FUNCTION_BLOCK PICKER_MODEL_NO_SFC_VIEW (* Composite Function Block Type *)
  (* Standard: 61499-2 *)
  (* Version 0.2, 2003-12-05, JHC, Rockwell Automation, Renamed from NEWCOMPFB. *)
  (* Version 0.1, 2002-01-08, JHC, Rockwell Automation, Added DLY FB as example. *)
  (* Version 0.0, 2000-05-27, JHC, Rockwell Automation *)
  (* Compiler header: package fb.rt.pnp; *)
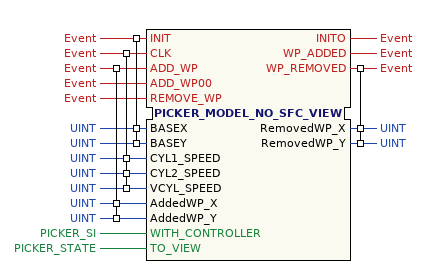
  EVENT_INPUT
    INIT WITH BASEX, BASEY; (* Initialisation *)
    CLK WITH CYL1_SPEED, CYL2_SPEED, VCYL_SPEED;
    ADD_WP WITH AddedWP_X, AddedWP_Y;
    ADD_WP00;
    REMOVE_WP;
  END_EVENT
  EVENT_OUTPUT
    INITO; (* Initialization Confirm *)
    WP_ADDED;
    WP_REMOVED WITH RemovedWP_X, RemovedWP_Y;
  END_EVENT
  VAR_INPUT
    BASEX : UINT;
    BASEY : UINT;
    CYL1_SPEED : UINT;
    CYL2_SPEED : UINT;
    VCYL_SPEED : UINT;
    AddedWP_X : UINT;
    AddedWP_Y : UINT;
  END_VAR
  VAR_OUTPUT
    RemovedWP_X : UINT;
    RemovedWP_Y : UINT;
  END_VAR
  SOCKETS
    WITH_CONTROLLER : PICKER_SI;
    TO_VIEW : PICKER_STATE;
  END_SOCKETS
  FBS
    MODEL : Model;
    s11 : my_sensor(ZONE := [305,310]);
    s12 : my_sensor(ZONE := [381,385]);
    s13 : my_sensor(ZONE := [455,460]);
    s14 : my_sensor(ZONE := [535,540]);
    Machado_SFC : MachadoSFC;
  END_FBS
  EVENT_CONNECTIONS
    INIT TO MODEL.INIT;
    MODEL.INITO TO TO_VIEW.INIT;
    MODEL.INITO TO INITO;
    MODEL.CNF TO WITH_CONTROLLER.CNF;
    WITH_CONTROLLER.REQ TO MODEL.REQ;
    CLK TO MODEL.CLK;
    ADD_WP TO MODEL.ADD_WP;
    REMOVE_WP TO MODEL.REMOVE_WP;
    MODEL.WP_ADDED TO WP_ADDED;
    MODEL.WP_REMOVED TO WP_REMOVED;
    MODEL.INITO TO s11.INIT;
    s11.INITO TO s12.INIT;
    s12.INITO TO s13.INIT;
    s13.INITO TO s14.INIT;
    MODEL.CNF TO s11.REQ;
    MODEL.CNF TO s12.REQ;
    MODEL.CNF TO s13.REQ;
    MODEL.CNF TO s14.REQ;
    s11.CNF TO WITH_CONTROLLER.CNF;
    s12.CNF TO WITH_CONTROLLER.CNF;
    s13.CNF TO WITH_CONTROLLER.CNF;
    s14.CNF TO WITH_CONTROLLER.CNF;
    ADD_WP00 TO MODEL.ADD_WP00;
    s14.INITO TO Machado_SFC.INIT;
    MODEL.CHG TO Machado_SFC.REQ;
    MODEL.CHG TO WITH_CONTROLLER.CNF;
    MODEL.CNF TO TO_VIEW.CHG;
    s11.CNF TO Machado_SFC.REQ;
    s12.CNF TO Machado_SFC.REQ;
    s13.CNF TO Machado_SFC.REQ;
    s14.CNF TO Machado_SFC.REQ;
    Machado_SFC.CNF TO MODEL.CYL_IND;
  END_CONNECTIONS
  DATA_CONNECTIONS
    MODEL.BASE_X TO TO_VIEW.BASE_X;
    MODEL.BASE_Y TO TO_VIEW.BASE_Y;
    MODEL.CYL1_X TO TO_VIEW.CYL1_X;
    MODEL.CYL1_Y TO TO_VIEW.CYL1_Y;
    MODEL.CYL2_X TO TO_VIEW.CYL2_X;
    MODEL.CYL2_Y TO TO_VIEW.CYL2_Y;
    MODEL.VCYL_X TO TO_VIEW.VCYL_X;
    MODEL.VCYL_Y TO TO_VIEW.VCYL_Y;
    MODEL.WP_X TO TO_VIEW.WP1_X;
    MODEL.WP_Y TO TO_VIEW.WP1_Y;
    MODEL.VACUUM_ON TO TO_VIEW.VACUUM_ON;
    BASEX TO MODEL.BASEX;
    BASEY TO MODEL.BASEY;
    CYL1_SPEED TO MODEL.CYL1_SPEED;
    CYL2_SPEED TO MODEL.CYL2_SPEED;
    VCYL_SPEED TO MODEL.VCYL_SPEED;
    MODEL.vchome TO WITH_CONTROLLER.vchome;
    MODEL.vcend TO WITH_CONTROLLER.vcend;
    AddedWP_X TO MODEL.AddedWP_X;
    AddedWP_Y TO MODEL.AddedWP_Y;
    MODEL.RemovedWP_X TO RemovedWP_X;
    MODEL.RemovedWP_Y TO RemovedWP_Y;
    MODEL.VCYL_X TO s11.POS;
    MODEL.VCYL_X TO s12.POS;
    MODEL.VCYL_X TO s13.POS;
    MODEL.VCYL_X TO s14.POS;
    s11.VALUE TO WITH_CONTROLLER.S11;
    s12.VALUE TO WITH_CONTROLLER.S12;
    s13.VALUE TO WITH_CONTROLLER.S13;
    s14.VALUE TO WITH_CONTROLLER.S14;
    MODEL.WP3_X TO TO_VIEW.WP3_X;
    MODEL.WP3_Y TO TO_VIEW.WP3_Y;
    MODEL.WP2_X TO TO_VIEW.WP2_X;
    MODEL.WP2_Y TO TO_VIEW.WP2_Y;
    WITH_CONTROLLER.add1 TO MODEL.Add1;
    WITH_CONTROLLER.add2 TO MODEL.Add2;
    WITH_CONTROLLER.add3 TO MODEL.Add3;
    s11.VALUE TO Machado_SFC.s10;
    s12.VALUE TO Machado_SFC.s11;
    s13.VALUE TO Machado_SFC.s12;
    s14.VALUE TO Machado_SFC.s13;
    MODEL.vchome TO Machado_SFC.vcu;
    MODEL.vcend TO Machado_SFC.vcd;
    MODEL.VACUUM_ON TO Machado_SFC.vacuum;
    Machado_SFC.c1_front TO MODEL.cyl1_fwd;
    Machado_SFC.c1_back TO MODEL.cyl1_back;
    Machado_SFC.c2_front TO MODEL.cyl2_fwd;
    Machado_SFC.c2_back TO MODEL.cyl2_back;
    Machado_SFC.vc_down TO MODEL.vcyl_down;
    Machado_SFC.venturi_on TO MODEL.vacuum_on;
    Machado_SFC.venturi_off TO MODEL.vacuum_off;
    MODEL.VACUUM_ON TO WITH_CONTROLLER.wp_sucked_in;
    MODEL.pp0 TO WITH_CONTROLLER.wp11;
    MODEL.pp1 TO WITH_CONTROLLER.wp12;
    MODEL.pp2 TO WITH_CONTROLLER.wp13;
    MODEL.pp3 TO WITH_CONTROLLER.wp14;
    MODEL.pp0 TO Machado_SFC.pp0;
    MODEL.pp1 TO Machado_SFC.pp1;
    MODEL.pp2 TO Machado_SFC.pp2;
    MODEL.pp3 TO Machado_SFC.pp3;
  END_CONNECTIONS
END_FUNCTION_BLOCK
